TYPE ST_PowerGroupOutImm :
STRUCT
    Status     : ST_PowerGroupStatus;
END_STRUCT
END_TYPE

(* stored: Version 1.1.0.1, ProductVersion 3.1.4024.12
   DUT ST_PowerGroupOutImm: Id {c972c0cb-3543-4263-a319-8d76a582a386} *)
